(* IEC 61131-3 sources: conversion/src, 14 files *)

(* ---- ConversionMode.st ---- *)
NAMESPACE Simatic.Ax.Conversion
    TYPE
        ConversionMode : WORD (NONE := WORD#16#0000, FORCE_SIGN := WORD#16#0001) := NONE;
    END_TYPE
END_NAMESPACE

(* ---- AnyIntToString.st ---- *)
USING System.Strings;
USING System.Math;

NAMESPACE Simatic.Ax.Conversion
    FUNCTION INTERNAL AnyIntToString : STRING
        VAR_INPUT
            value : LINT;
            mode : ConversionMode := ConversionMode#NONE;
        END_VAR
        VAR_TEMP
            _value : LINT;
            digit : INT;
            c : USINT;
            i : INT;
            digits : INT;
            offset : INT;
            s : STRING[1];
            t : ARRAY[0..19] OF CHAR; // MAX: -9223372036854775808
        END_VAR

        _value := value;
        digits := CountDigits(value);
        IF (_value < 0) THEN  // Add sign to
            AnyIntToString := Concat(AnyIntToString, '-');
            offset := 1; // keep space for the sign
        ELSIF (_value > 0 AND (mode AND ConversionMode#FORCE_SIGN) = ConversionMode#FORCE_SIGN) THEN  // Add sign to
            AnyIntToString := Concat(AnyIntToString, '+');
            offset := 1; // keep space for the sign
        ELSE
            offset := 0;
        END_IF;

        FOR i := 0 TO digits - 1 DO
            digit := ABS(TO_INT(_value MOD 10));
            c := TO_USINT('0') + TO_USINT(digit);
            t[digits - i - 1] := TO_CHAR(TO_BYTE(c));
            _value := _value / 10;
        END_FOR;
        FOR i := 0 TO digits - 1 DO
            s[1] := t[i];
            AnyIntToString := Concat(AnyIntToString, s);
        END_FOR;
    END_FUNCTION

    FUNCTION INTERNAL ULintToString : STRING
        VAR_INPUT
            value : ULINT;
            mode : ConversionMode := ConversionMode#NONE;
        END_VAR
        VAR_TEMP
            _value : ULINT;
            digit : INT;
            c : USINT;
            i : INT;
            digits : INT;
            offset : INT;
            s : STRING[1];
            t : ARRAY[0..19] OF CHAR; // MAX: -9223372036854775808
        END_VAR

        _value := value;
        // Prepare the sting with the correct lenght
        digits := CountDigits(value);

        IF (_value > ULINT#0 AND (mode AND ConversionMode#FORCE_SIGN) = ConversionMode#FORCE_SIGN) THEN  // Add sign to
            ULintToString[1] := '+';
            offset := 1; // keep space for the sign
        ELSE
            offset := 0;
        END_IF;

        FOR i := 0 TO digits - 1 DO
            digit := ABS(TO_INT(_value MOD UINT#10));
            c := TO_USINT('0') + TO_USINT(digit);
            t[digits - i - 1] := TO_CHAR(TO_BYTE(c));
            _value := _value / UINT#10;
        END_FOR;
        FOR i := 0 TO digits - 1 DO
            s[1] := t[i];
            ULintToString := Concat(ULintToString, s);
        END_FOR;
    END_FUNCTION
END_NAMESPACE

(* ---- ArrayToString.st ---- *)
USING System.Strings;

NAMESPACE Simatic.Ax.Conversion.Arrays
    // add a new comment
    FUNCTION ToString : STRING
        VAR_INPUT
            arr : ARRAY[*] OF CHAR;
            startIdx : INT;
            endIdx : INT;
        END_VAR
        VAR CONSTANT
            MAX_STR_LEN : INT := 254;
        END_VAR
        VAR_TEMP
            i : DINT;
            _lb : DINT;
            _ub : DINT;
            _arrayLen : DINT;
        END_VAR
        _lb := LOWER_BOUND(arr, 1);
        _ub := UPPER_BOUND(arr, 1);

        // start index > end index
        IF (startIdx > endIdx) THEN
            ToString := '';
            RETURN;
        END_IF;

        // start index is not existing
        IF (startIdx < _lb) OR (startIdx > _ub) AND (startIdx <> 0) THEN
            ToString := '';
            RETURN;
        END_IF;
        // end index is ot existing
        IF (endIdx > _ub) THEN
            ToString := '';
            RETURN;
        END_IF;
        _arrayLen := endIdx - startIdx + 1;

        IF (_arrayLen > MAX_STR_LEN) THEN
            _arrayLen := MAX_STR_LEN;
        END_IF;

        FOR i := 0 TO _arrayLen - 1 DO
            ToString[i + 1] := arr[i + _lb + startIdx];
        END_FOR;

    END_FUNCTION

    FUNCTION ToString : STRING
        VAR_INPUT
            arr : ARRAY[*] OF CHAR;
        END_VAR
        VAR CONSTANT
            MAX_STR_LEN : INT := 254;
        END_VAR
        VAR_TEMP
            i : DINT;
            _lb : DINT;
            _ub : DINT;
            _arrayLen : DINT;
        END_VAR
        _lb := LOWER_BOUND(arr, 1);
        _ub := UPPER_BOUND(arr, 1);

        _arrayLen := _ub - _lb + 1;

        IF (_arrayLen > MAX_STR_LEN) THEN
            _arrayLen := MAX_STR_LEN;
        END_IF;

        FOR i := 0 TO _arrayLen - 1 DO
            ToString[i + 1] := arr[i + _lb];
        END_FOR;

    END_FUNCTION
END_NAMESPACE

(* ---- CountDigits.st ---- *)
USING System.Math;

NAMESPACE Simatic.Ax.Conversion
    FUNCTION CountDigits : INT
        VAR_INPUT
            value : LINT;
        END_VAR
        VAR_TEMP
            divisor : LINT := LINT#1;
            i : INT;
        END_VAR
        VAR CONSTANT
            MAX_DIGITS : INT := 19;
        END_VAR

        IF (value = 0) THEN
            CountDigits := 1;
            RETURN;
        END_IF;

        FOR i := 0 TO MAX_DIGITS DO
            IF(value / divisor = 0) THEN
                CountDigits := i;
                RETURN;
            END_IF;
            divisor := divisor * 10;
        END_FOR;
        CountDigits := 19;
    END_FUNCTION
END_NAMESPACE

(* ---- CreateStringWithBlanksOfLength.st ---- *)
USING System.Strings;

NAMESPACE Simatic.Ax.Conversion
    FUNCTION CreateStringWithBlanksOfLength : STRING
        VAR_INPUT
            str : STRING;
            len : INT;
            _tempString : STRING[1] := '0';
        END_VAR
        VAR_TEMP
            i : INT;
        END_VAR
        CreateStringWithBlanksOfLength := '';

        FOR i := 1 TO len  DO
            CreateStringWithBlanksOfLength := Concat(CreateStringWithBlanksOfLength, _tempString);
        END_FOR;

    END_FUNCTION
END_NAMESPACE

(* ---- HexToString.st ---- *)
USING System;
USING System.Strings;

NAMESPACE Simatic.Ax.Conversion

    FUNCTION PUBLIC HTA : STRING
        VAR_INPUT
            b : BYTE;
        END_VAR
        VAR_TEMP
            tempS : STRING[2];
            tempN1 : BYTE;
            tempN2 : BYTE;
        END_VAR
        tempN1 := b AND BYTE#16#0F;
        tempN2 := SHR(b,USINT#4);

        HTA := Concat(LookUpHEX(tempN2),LookUpHEX(tempN1));

    END_FUNCTION

    FUNCTION LookUpHEX : CHAR
        VAR_INPUT
            nibble : BYTE;
        END_VAR
        VAR
            h : ARRAY[0..15] of CHAR := ['0','1','2','3','4','5','6','7','8','9','A','B','C','D','E','F'];
        END_VAR

        LookUpHEX := h[TO_UINT(nibble)];

    END_FUNCTION

END_NAMESPACE

(* ---- IntToString.st ---- *)
USING System.Strings;
USING System.Math;

NAMESPACE Simatic.Ax.Conversion.Integer
    FUNCTION ToString : STRING[4]
        VAR_INPUT
            value : SINT;
            mode : ConversionMode := ConversionMode#NONE;
        END_VAR
        VAR_TEMP
        END_VAR
        ToString := AnyIntToString(value := value, mode := mode);
    END_FUNCTION

    FUNCTION ToString : STRING[4]
        VAR_INPUT
            value : USINT;
            mode : ConversionMode := ConversionMode#NONE;
        END_VAR
        VAR_TEMP
        END_VAR
        ToString := AnyIntToString(value := value, mode := mode);
    END_FUNCTION

    FUNCTION ToString : STRING[6]
        VAR_INPUT
            value : INT;
            mode : ConversionMode := ConversionMode#NONE;
        END_VAR
        VAR_TEMP
        END_VAR
        ToString := AnyIntToString(value := value, mode := mode);
    END_FUNCTION

    FUNCTION ToString : STRING[6]
        VAR_INPUT
            value : UINT;
            mode : ConversionMode := ConversionMode#NONE;
        END_VAR
        VAR_TEMP
        END_VAR
        ToString := AnyIntToString(value := value, mode := mode);
    END_FUNCTION

    FUNCTION ToString : STRING[11]
        VAR_INPUT
            value : DINT;
            mode : ConversionMode := ConversionMode#NONE;
        END_VAR
        VAR_TEMP
        END_VAR
        ToString := AnyIntToString(value := value, mode := mode);
    END_FUNCTION

    FUNCTION ToString : STRING[11]
        VAR_INPUT
            value : UDINT;
            mode : ConversionMode := ConversionMode#NONE;
        END_VAR
        VAR_TEMP
        END_VAR
        ToString := AnyIntToString(value := value, mode := mode);
    END_FUNCTION

    FUNCTION ToString : STRING[20]
        VAR_INPUT
            value : LINT;
            mode : ConversionMode := ConversionMode#NONE;
        END_VAR
        VAR_TEMP
        END_VAR
        ToString := AnyIntToString(value := value, mode := mode);
    END_FUNCTION

    FUNCTION ToString : STRING[21]
        VAR_INPUT
            value : ULINT;
            mode : ConversionMode := ConversionMode#NONE;
        END_VAR
        VAR_TEMP
        END_VAR
        ToString := ULintToString(value := value, mode := mode);
    END_FUNCTION
END_NAMESPACE

(* ---- new_feature.st ---- *)
NAMESPACE Simatic.Ax.Conversion
    FUNCTION new_feature : Int
        VAR_INPUT
        END_VAR
        VAR_TEMP
        END_VAR

        ;
    END_FUNCTION
END_NAMESPACE

(* ---- SetStringLength.st ---- *)
USING System.Strings;

NAMESPACE Simatic.Ax.Conversion
    FUNCTION SetStringLength : STRING
        VAR_INPUT
            str : STRING;
            len : INT;
        END_VAR
        SetStringLength := '';

    END_FUNCTION
END_NAMESPACE

(* ---- StringToAnyInt.st ---- *)
USING System.Strings;

NAMESPACE Simatic.Ax.Conversion
    FUNCTION INTERNAL StringToAnyInt : BOOL
        VAR_INPUT
            str : STRING;
        END_VAR
        VAR_OUTPUT
            value : LINT;
        END_VAR
        VAR_TEMP
            _len : INT;
            i : INT;
            _val : INT;
            _sig : INT;
            _start : INT;
        END_VAR

        _len := LengthOf(str);

        IF (str[1] = '+') THEN
            _sig := 1;
            _start := 2;
        ELSIF (str[1] = '-') THEN
            _sig := -1;
            _start := 2;
        ELSE
            _sig := 1;
            _start := 1;
        END_IF;
        value := 0;
        FOR i := _start TO _len DO

            value := value * 10;
            CASE str[i] OF
                '0' : _val := 0;
                '1' : _val := 1;
                '2' : _val := 2;
                '3' : _val := 3;
                '4' : _val := 4;
                '5' : _val := 5;
                '6' : _val := 6;
                '7' : _val := 7;
                '8' : _val := 8;
                '9' : _val := 9;
                CHAR#0:
                    StringToAnyInt := TRUE;
                    value := value * _sig;
                    RETURN;
            ELSE
                value := 0;
                StringToAnyInt := FALSE;
                RETURN;
            END_CASE;
            value := value + _val;
        END_FOR;
        value := value * _sig;
        IF (_sig = 1 AND value < 0) OR (_sig = -1 AND value > 0) THEN
            value := 0;
            StringToAnyInt := FALSE;
        ELSE
            StringToAnyInt := TRUE;
        END_IF;
    END_FUNCTION

    FUNCTION INTERNAL StringToULint: BOOL
        VAR_INPUT
            str : STRING;
        END_VAR
        VAR_OUTPUT
            value : ULINT;
        END_VAR
        VAR_TEMP
            _len : INT;
            i : INT;
            _val : ULINT;
            _start : INT;
        END_VAR

        _len := LengthOf(str);

        IF (str[1] = '+') THEN
            _start := 2;
        ELSE
            _start := 1;
        END_IF;

        value := ULINT#0;

        FOR i := _start TO _len DO

            value := value * ULINT#10;
            CASE str[i] OF
                '0' : _val := ULINT#0;
                '1' : _val := ULINT#1;
                '2' : _val := ULINT#2;
                '3' : _val := ULINT#3;
                '4' : _val := ULINT#4;
                '5' : _val := ULINT#5;
                '6' : _val := ULINT#6;
                '7' : _val := ULINT#7;
                '8' : _val := ULINT#8;
                '9' : _val := ULINT#9;
                CHAR#0:
                StringToULint := TRUE;
                    RETURN;
            ELSE
                value := ULINT#0;
                StringToULint := FALSE;
                RETURN;
            END_CASE;
            value := value + _val;
        END_FOR;
        StringToULint := TRUE;
    END_FUNCTION
END_NAMESPACE

(* ---- StringToArray.st ---- *)
USING System.Strings;

NAMESPACE Simatic.Ax.Conversion.Strings
    FUNCTION ToArray : DINT
        VAR_INPUT
            str : STRING;
        END_VAR
        VAR_IN_OUT
            arr : ARRAY[*] OF CHAR;
        END_VAR
        VAR_TEMP
            i : DINT;
            _lb : DINT;
            _ub : DINT;
            _maxLen : DINT;
        END_VAR
        _lb := LOWER_BOUND(arr, 1);
        _ub := UPPER_BOUND(arr, 1);
        _maxLen := LengthOf(str);

        IF (_maxLen > _ub - _lb + 1) THEN
            _maxLen := TO_INT(_ub - _lb + 1);
        END_IF;

        FOR i := 0 TO _maxLen - 1 DO
            arr[i + _lb] := str[i + 1];
        END_FOR;
        ToArray := i;
    END_FUNCTION
END_NAMESPACE

(* ---- StringToArrayOfInt.st ---- *)
USING System.Strings;

NAMESPACE Simatic.Ax.Conversion

    FUNCTION INTERNAL StringToArrayOfLint : BOOL
        VAR_INPUT
            str: STRING;
        END_VAR
        VAR_IN_OUT
            arr: ARRAY[*] OF LINT;
        END_VAR
        VAR_TEMP
            arrayStart: INT;
            arrayEnd: INT;
            lb: DINT;
            ub: DINT;
            index: INT;
            intString: STRING;
            arrayIndex: DINT;

            elementStart: INT;
            elementEnd: INT;
            inElement: BOOL := FALSE;
            elementFound: BOOL := FALSE;

            substr: STRING;
            parseSucces: BOOL;
            value: LINT; //mehr möglich machen!
        END_VAR

        StringToArrayOfLint := FALSE;
        IF LengthOf(str) = 0 THEN
            RETURN;
        END_IF;

        //TODO: make funktion out of it that gives back boundaries
        lb := LOWER_BOUND(arr, 1);
        ub := UPPER_BOUND(arr, 1);

    FOR index := 1 TO LengthOf(str) DO
        IF str[index] = '[' THEN
            arrayStart := index + 1;
            EXIT;
        END_IF;
    END_FOR;

    FOR index := LengthOf(str) TO 1 BY -1 DO
        IF str[index] = ']' THEN
            arrayEnd := index;
            EXIT;
        END_IF;
    END_FOR;

    arrayIndex := LOWER_BOUND(arr, 1);
    //loop through string
    FOR index := arrayStart TO arrayEnd DO

        IF NOT inElement AND NOT ((str[index] = ' ' OR str[index] = ',')) THEN
            elementStart := index;
            inElement := TRUE;
        END_IF;

        IF inElement AND (str[index] = ' ' OR str[index] = ',' OR str[index] = ']') THEN
            elementEnd := index;
            inElement := FALSE;
            elementFound := TRUE;
        END_IF;

        //substring
        IF elementFound THEN
            substr := Substring(str, elementStart, elementEnd - elementStart);
            parseSucces := StringToAnyInt(substr, value);
            IF parseSucces THEN
                arr[arrayIndex] := value;
                arrayIndex := arrayIndex + 1;
                elementFound := FALSE;
                StringToArrayOfLint := TRUE;
            ELSE
                StringToArrayOfLint := FALSE;
                RETURN;
            END_IF;
        END_IF;
    END_FOR;

    END_FUNCTION

END_NAMESPACE

(* ---- ToInt.st ---- *)
USING System.Strings;

NAMESPACE Simatic.Ax.Conversion.Strings
    FUNCTION ToInt : BOOL
        VAR_INPUT
            str : STRING;
        END_VAR
        VAR_OUTPUT
            value : SINT;
        END_VAR
        VAR_TEMP
            _val : LINT;
        END_VAR
        VAR CONSTANT
            MAX_VAL : LINT := LINT#127;
            MIN_VAL : LINT := LINT#-128;
        END_VAR

        ToInt := StringToAnyInt(str := str, value => _val);

        IF (_val < MIN_VAL) OR (_val > MAX_VAL) THEN
            value := SINT#0;
            ToInt := FALSE;
        ELSE
            value := TO_SINT(_val);
        END_IF;
    END_FUNCTION

    FUNCTION ToInt : BOOL
        VAR_INPUT
            str : STRING;
        END_VAR
        VAR_OUTPUT
            value : INT;
        END_VAR
        VAR_TEMP
            _val : LINT;
        END_VAR
        VAR CONSTANT
            MAX_VAL : LINT := LINT#32767;
            MIN_VAL : LINT := LINT#-32768;
        END_VAR

        ToInt := StringToAnyInt(str := str, value => _val);

        IF (_val < MIN_VAL) OR (_val > MAX_VAL) THEN
            value := SINT#0;
            ToInt := FALSE;
        ELSE
            value := TO_INT(_val);
        END_IF;
    END_FUNCTION

    FUNCTION ToInt : BOOL
        VAR_INPUT
            str : STRING;
        END_VAR
        VAR_OUTPUT
            value : DINT;
        END_VAR
        VAR_TEMP
            _val : LINT;
        END_VAR
        VAR CONSTANT
            MAX_VAL : LINT := LINT#2147483647;
            MIN_VAL : LINT := LINT#-2147483648;
        END_VAR

        ToInt := StringToAnyInt(str := str, value => _val);

        IF (_val < MIN_VAL) OR (_val > MAX_VAL) THEN
            value := SINT#0;
            ToInt := FALSE;
        ELSE
            value := TO_DINT(_val);
        END_IF;
    END_FUNCTION

    FUNCTION ToInt : BOOL
        VAR_INPUT
            str : STRING;
        END_VAR
        VAR_OUTPUT
            value : LINT;
        END_VAR
        VAR_TEMP
            _val : LINT;
        END_VAR
        VAR CONSTANT
            MAX_VAL : LINT := LINT#9223372036854775807;
            MIN_VAL : LINT := LINT#-9223372036854775808;
        END_VAR

        ToInt := StringToAnyInt(str := str, value => _val);

        IF (_val < MIN_VAL) OR (_val > MAX_VAL) THEN
            value := SINT#0;
            ToInt := FALSE;
        ELSE
            value := _val;
        END_IF;
    END_FUNCTION

    FUNCTION ToInt : BOOL
        VAR_INPUT
            str : STRING;
        END_VAR
        VAR_OUTPUT
            value : USINT;
        END_VAR
        VAR_TEMP
            _val : LINT;
        END_VAR
        VAR CONSTANT
            MAX_VAL : LINT := LINT#255;
            MIN_VAL : LINT := LINT#0;
        END_VAR

        ToInt := StringToAnyInt(str := str, value => _val);

        IF (_val < MIN_VAL) OR (_val > MAX_VAL) THEN
            value := USINT#0;
            ToInt := FALSE;
        ELSE
            value := TO_USINT(_val);
        END_IF;
    END_FUNCTION

    FUNCTION ToInt : BOOL
        VAR_INPUT
            str : STRING;
        END_VAR
        VAR_OUTPUT
            value : UINT;
        END_VAR
        VAR_TEMP
            _val : LINT;
        END_VAR
        VAR CONSTANT
            MAX_VAL : LINT := LINT#65535;
            MIN_VAL : LINT := LINT#0;
        END_VAR

        ToInt := StringToAnyInt(str := str, value => _val);

        IF (_val < MIN_VAL) OR (_val > MAX_VAL) THEN
            value := USINT#0;
            ToInt := FALSE;
        ELSE
            value := TO_UINT(_val);
        END_IF;
    END_FUNCTION

    FUNCTION ToInt : BOOL
        VAR_INPUT
            str : STRING;
        END_VAR
        VAR_OUTPUT
            value : UDINT;
        END_VAR
        VAR_TEMP
            _val : LINT;
        END_VAR
        VAR CONSTANT
            MAX_VAL : LINT := LINT#4294967295;
            MIN_VAL : LINT := LINT#0;
        END_VAR

        ToInt := StringToAnyInt(str := str, value => _val);

        IF (_val < MIN_VAL) OR (_val > MAX_VAL) THEN
            value := USINT#0;
            ToInt := FALSE;
        ELSE
            value := TO_UDINT(_val);
        END_IF;
    END_FUNCTION

END_NAMESPACE

(* ---- TRUNC.st ---- *)
NAMESPACE Simatic.Ax.Conversion

    /// Truncates a 64-bit floating-point number (LREAL) to an integer.
    ///
    /// This function truncates the input LREAL value to the nearest integer toward zero.
    /// It handles both positive and negative values.
    ///
    /// @param Value The LREAL value to truncate.
    /// @return The truncated integer value.
    {axcode:docs-v0:@simatic-ax/conversion:TRUNC.md}
    FUNCTION TRUNC : DINT
        VAR_INPUT
            Value : LREAL;
        END_VAR
        TRUNC := TO_DINT(Value);
        IF Value > 0.0 THEN
            IF TO_LREAL(TRUNC) > Value THEN
                TRUNC := TRUNC - 1;
            END_IF;
        ELSE
            IF TO_LREAL(TRUNC) < Value THEN
                TRUNC := TRUNC + 1;
            END_IF;
        END_IF;
    END_FUNCTION

    /// Truncates a 32-bit floating-point number (REAL) to an integer.
    ///
    /// This function truncates the input REAL value to the nearest integer toward zero.
    /// It handles both positive and negative values.
    ///
    /// @param Value The REAL value to truncate.
    /// @return The truncated integer value.
    {axcode:docs-v0:@simatic-ax/conversion:TRUNC.md}
    FUNCTION TRUNC : DINT
        VAR_INPUT
            Value : REAL;
        END_VAR
        TRUNC := TO_DINT(Value);
        IF Value > 0.0 THEN
            IF TO_LREAL(TRUNC) > Value THEN
                TRUNC := TRUNC - 1;
            END_IF;
        ELSE
            IF TO_LREAL(TRUNC) < Value THEN
                TRUNC := TRUNC + 1;
            END_IF;
        END_IF;
    END_FUNCTION

END_NAMESPACE
